Yaskawa INFORM job: TROCA_CAPA.JBI

/JOB
//NAME TROCA_CAPA
///FOLDERNAME SERVICO
//POS
///NPOS 0,0,0,0,0,0
//INST
///DATE 2022/06/11 12:10
///ATTR SC,RW
///GROUP1 RB1,ST1
NOP
END
